(* IEC 61131-3 sources: AXOpen/src/integrations/ctrl/src/IntegrationTests/data, 3 files *)

(* ---- AxoDataFragmentExchange.st ---- *)
USING AXOpen.Core;
USING AXOpen.Data;
USING AXOpen.Probers;

NAMESPACE IntegrationAxoDataFramentsExchange

    CLASS AxoDataFragmentExchangeContext EXTENDS AXOpen.Core.AxoContext
        VAR PUBLIC
            PD : ProcessData;
            CreateTest : DataCreateTest;
            ReadTest : DataReadTest;
            UpdateTest : DataUpdateTest;
            DeleteTest : DataDeleteTest;
        END_VAR

        METHOD PROTECTED OVERRIDE Main

            PD.Run(THIS);

            CreateTest.InjectManger(PD);
            CreateTest.Run(THIS);

            ReadTest.InjectManger(PD);
            ReadTest.Run(THIS);

            DeleteTest.InjectManger(PD);
            DeleteTest.Run(THIS);

            UpdateTest.InjectManger(PD);
            UpdateTest.Run(THIS);
        END_METHOD

    END_CLASS

    CLASS ProcessData EXTENDS AXOpen.Data.AxoDataFragmentExchange
        VAR PUBLIC
            {#ix-attr:[AXOpen.Data.AxoDataFragmentAttribute]}
            Set : SharedProductionDataManager;
            {#ix-attr:[AXOpen.Data.AxoDataFragmentAttribute]}
            Manip : FragmentProcessDataManger;
        END_VAR
    END_CLASS

    CLASS SharedProductionData EXTENDS AXOpen.Data.AxoDataEntity
        VAR PUBLIC
            ComesFrom : INT;
            GoesTo : INT;
        END_VAR
    END_CLASS

    CLASS SharedProductionDataManager EXTENDS AXOpen.Data.AxoDataExchange
        VAR PUBLIC
            {#ix-generic:TOnline}
            {#ix-generic:TPlain as POCO}
            {#ix-attr:[AXOpen.Data.AxoDataEntityAttribute]}
            {#ix-attr:[Container(Layout.Stack)]}
            Set : SharedProductionData;
        END_VAR
    END_CLASS

    CLASS FragmentProcessDataManger
        EXTENDS AXOpen.Data.AxoDataExchange
        VAR PUBLIC
            {#ix-generic:TOnline}
            {#ix-generic:TPlain as POCO}
            {#ix-attr:[AXOpen.Data.AxoDataEntityAttribute]}
            {#ix-attr:[Container(Layout.Stack)]}
            Set : FragmentProcessData;
        END_VAR
    END_CLASS

    CLASS FragmentProcessData
        EXTENDS AXOpen.Data.AxoDataEntity
        VAR PUBLIC
            CounterDelay : ULINT;
        END_VAR
    END_CLASS

    CLASS DataCreateTest EXTENDS AxoProberWithCompletedCondition
        VAR PUBLIC
            Manager : IAxoDataExchange;
            Identifier : STRING[254];
        END_VAR
        METHOD PROTECTED OVERRIDE Test : BOOL
            VAR
                _taskState : IAxoTaskState;
            END_VAR
            IF(Manager <> NULL) THEN
                _taskState := Manager.Create(Identifier);
                THIS.ThrowWhen(_taskState.HasError(), _taskState.GetErrorDetails());
                Test := _taskState.IsDone();
            END_IF;
        END_METHOD

        METHOD OVERRIDE OnRestore
            SUPER.OnRestore();
            IF(Manager <> NULL) THEN
                 Manager.Restore();
            END_IF;
        END_METHOD

        METHOD PUBLIC InjectManger
            VAR_INPUT
                Injectee : IAxoDataExchange;
            END_VAR
            Manager := Injectee;
        END_METHOD
    END_CLASS

    CLASS DataReadTest EXTENDS AxoProberWithCompletedCondition
        VAR PUBLIC
            Manager : IAxoDataExchange;
            Identifier : STRING[254];
        END_VAR
        METHOD PROTECTED OVERRIDE Test : BOOL
            VAR
                _taskState : IAxoTaskState;
            END_VAR
            IF(Manager <> NULL) THEN
                _taskState := Manager.Read(Identifier);
                THIS.ThrowWhen(_taskState.HasError(), _taskState.GetErrorDetails());
                Test := _taskState.IsDone();
            END_IF;
        END_METHOD

        METHOD OVERRIDE OnRestore
            SUPER.OnRestore();
            IF(Manager <> NULL) THEN
                 Manager.Restore();
            END_IF;
        END_METHOD

        METHOD PUBLIC InjectManger
            VAR_INPUT
                Injectee : IAxoDataExchange;
            END_VAR
            Manager := Injectee;
        END_METHOD
    END_CLASS

    CLASS DataUpdateTest EXTENDS AxoProberWithCompletedCondition
        VAR PUBLIC
            Manager : IAxoDataExchange;
            Identifier : STRING[254];
        END_VAR
        METHOD PROTECTED OVERRIDE Test : BOOL
            VAR
                _taskState : IAxoTaskState;
            END_VAR
            IF(Manager <> NULL) THEN
                _taskState := Manager.Update(Identifier);
                THIS.ThrowWhen(_taskState.HasError(), _taskState.GetErrorDetails());
                Test := _taskState.IsDone();
            END_IF;
        END_METHOD

        METHOD OVERRIDE OnRestore
            SUPER.OnRestore();
            IF(Manager <> NULL) THEN
                 Manager.Restore();
            END_IF;
        END_METHOD

        METHOD PUBLIC InjectManger
            VAR_INPUT
                Injectee : IAxoDataExchange;
            END_VAR
            Manager := Injectee;
        END_METHOD
    END_CLASS

    CLASS DataDeleteTest EXTENDS AxoProberWithCompletedCondition
        VAR PUBLIC
            Manager : IAxoDataExchange;
            Identifier : STRING[254];
        END_VAR
        METHOD PROTECTED OVERRIDE Test : BOOL
            VAR
                _taskState : IAxoTaskState;
            END_VAR
            IF(Manager <> NULL) THEN
                _taskState := Manager.Delete(Identifier);
                THIS.ThrowWhen(_taskState.HasError(), _taskState.GetErrorDetails());
                Test := _taskState.IsDone();
            END_IF;
        END_METHOD

        METHOD OVERRIDE OnRestore
            SUPER.OnRestore();
            IF(Manager <> NULL) THEN
                 Manager.Restore();
            END_IF;
        END_METHOD

        METHOD PUBLIC InjectManger
            VAR_INPUT
                Injectee : IAxoDataExchange;
            END_VAR
            Manager := Injectee;
        END_METHOD
    END_CLASS
END_NAMESPACE

(* ---- DataExchangeLightTests.st ---- *)
USING ix.framework.core;
USING ix.framework.data;
USING ix.framework.probers;

NAMESPACE IntegrationLightDirect
    CLASS DataExchangeLightTestsContext EXTENDS IxContext
        VAR PUBLIC
            DM : IDataExchange;
            CreateTest : DataCreateTest;
            ReadTest : DataReadTest;
            UpdateTest : DataUpdateTest;
            DeleteTest : DataDeleteTest;
        END_VAR

        METHOD PUBLIC InjectDM
            VAR_INPUT
                iDM : IDataExchange;
            END_VAR
            DM := iDM;
        END_METHOD

        METHOD PROTECTED OVERRIDE Main
            CreateTest.InjectManger(DM);
            CreateTest.Run(THIS);

            ReadTest.InjectManger(DM);
            ReadTest.Run(THIS);

            DeleteTest.InjectManger(DM);
            DeleteTest.Run(THIS);

            UpdateTest.InjectManger(DM);
            UpdateTest.Run(THIS);

        END_METHOD
    END_CLASS

    CLASS DataCreateTest EXTENDS ProberWithCompletedCondition
        VAR PUBLIC
            Manager : IDataExchange;
            Identifier : STRING[254];
        END_VAR
        METHOD PROTECTED OVERRIDE Test : BOOL
            VAR
                _taskState : IIxTaskState;
            END_VAR
            IF(Manager <> NULL) THEN
                _taskState := Manager.Create(Identifier);
                THIS.ThrowWhen(_taskState.HasError(), _taskState.GetErrorDetails());
                Test := _taskState.IsDone();
            END_IF;
        END_METHOD

        METHOD OVERRIDE OnRestore
            SUPER.OnRestore();
            IF(Manager <> NULL) THEN
                 Manager.Restore();
            END_IF;
        END_METHOD

        METHOD PUBLIC InjectManger
            VAR_INPUT
                Injectee : IDataExchange;
            END_VAR
            Manager := Injectee;
        END_METHOD
    END_CLASS

    CLASS DataReadTest EXTENDS ProberWithCompletedCondition
        VAR PUBLIC
            Manager : IDataExchange;
            Identifier : STRING[254];
        END_VAR
        METHOD PROTECTED OVERRIDE Test : BOOL
            VAR
                _taskState : IIxTaskState;
            END_VAR
            IF(Manager <> NULL) THEN
                _taskState := Manager.Read(Identifier);
                THIS.ThrowWhen(_taskState.HasError(), _taskState.GetErrorDetails());
                Test := _taskState.IsDone();
            END_IF;
        END_METHOD

        METHOD OVERRIDE OnRestore
            SUPER.OnRestore();
            IF(Manager <> NULL) THEN
                 Manager.Restore();
            END_IF;
        END_METHOD

        METHOD PUBLIC InjectManger
            VAR_INPUT
                Injectee : IDataExchange;
            END_VAR
            Manager := Injectee;
        END_METHOD
    END_CLASS

    CLASS DataUpdateTest EXTENDS ProberWithCompletedCondition
        VAR PUBLIC
            Manager : IDataExchange;
            Identifier : STRING[254];
        END_VAR
        METHOD PROTECTED OVERRIDE Test : BOOL
            VAR
                _taskState : IIxTaskState;
            END_VAR
            IF(Manager <> NULL) THEN
                _taskState := Manager.Update(Identifier);
                THIS.ThrowWhen(_taskState.HasError(), _taskState.GetErrorDetails());
                Test := _taskState.IsDone();
            END_IF;
        END_METHOD

        METHOD OVERRIDE OnRestore
            SUPER.OnRestore();
            IF(Manager <> NULL) THEN
                 Manager.Restore();
            END_IF;
        END_METHOD

        METHOD PUBLIC InjectManger
            VAR_INPUT
                Injectee : IDataExchange;
            END_VAR
            Manager := Injectee;
        END_METHOD
    END_CLASS

    CLASS DataDeleteTest EXTENDS ProberWithCompletedCondition
        VAR PUBLIC
            Manager : IDataExchange;
            Identifier : STRING[254];
        END_VAR
        METHOD PROTECTED OVERRIDE Test : BOOL
            VAR
                _taskState : IIxTaskState;
            END_VAR
            IF(Manager <> NULL) THEN
                _taskState := Manager.Delete(Identifier);
                THIS.ThrowWhen(_taskState.HasError(), _taskState.GetErrorDetails());
                Test := _taskState.IsDone();
            END_IF;
        END_METHOD

        METHOD OVERRIDE OnRestore
            SUPER.OnRestore();
            IF(Manager <> NULL) THEN
                 Manager.Restore();
            END_IF;
        END_METHOD

        METHOD PUBLIC InjectManger
            VAR_INPUT
                Injectee : IDataExchange;
            END_VAR
            Manager := Injectee;
        END_METHOD
    END_CLASS

    CLASS DataManager EXTENDS ix.framework.data.DataExchange
        VAR PUBLIC
            {#ix-attr:[DataEntityAttribute]}
            _data       : DataSet;
        END_VAR
    END_CLASS

    CLASS DataSet EXTENDS ix.framework.data.DataEntity
        VAR PUBLIC
            SomeData : STRING;
        END_VAR
    END_CLASS

END_NAMESPACE

(* ---- DataExchangeTest.st ---- *)
USING ix.framework.core;
USING ix.framework.data;
USING ix.framework.probers;

NAMESPACE IntegrationTests
    CLASS DataExchangeTestsContext EXTENDS IxContext
        VAR PUBLIC
            Create : DataExchangeCreateTest;
        END_VAR

        METHOD PROTECTED OVERRIDE Main
            Create.Initialize(THIS);
            Create.Run();
        END_METHOD
    END_CLASS

    CLASS DataExchangeCreateTest EXTENDS ProberWithCompletedCondition
        VAR PUBLIC
            Manager : DataExchangeManager;
            Identifier : STRING[254];
        END_VAR
        METHOD PROTECTED OVERRIDE Test : BOOL
            Manager.Initialize(THIS);
            Test := Manager.Create(Identifier).IsDone();
            Manager.Run();
            THIS.ThrowWhen(Manager.CreateTask.Status = eIxTaskState#Error);
            THIS.FailureDescription := Manager.CreateTask.ExceptionMessage;
        END_METHOD

        METHOD OVERRIDE OnRestore
            SUPER.OnRestore();
            Manager.Restore();
        END_METHOD
    END_CLASS

    CLASS DataExchangeManager EXTENDS DataExchange
        VAR PUBLIC
            _data       : DataSet;
        END_VAR
    END_CLASS

    CLASS DataSet EXTENDS DataEntity
        VAR PUBLIC
            SomeData : STRING;
        END_VAR
    END_CLASS
END_NAMESPACE
